// TIA Portal V17 export
// export: Created 2023-02-14T02:49:31.079512Z, ExportSetting WithDefaults, DisplayName Totally Integrated Automation Portal, DisplayVersion V17, DisplayName TIA Portal Openness, DisplayVersion V17, DisplayName TIA Portal Teamcenter Gateway, DisplayVersion V17, DisplayName TIA Portal Version Control Interface, DisplayVersion V17, DisplayName SINAMICS Startdrive Advanced, DisplayVersion V17, DisplayName SINAMICS Startdrive G130, G150, S120, S150, SINAMICS MV, S210, DisplayVersion V17, DisplayName SINAMICS Startdrive G110M, G120, G120C, G120D, G120P, G115D, DisplayVersion V17, DisplayName STEP 7 Professional, DisplayVersion V17, DisplayName STEP 7 Safety, DisplayVersion V17, DisplayName WinCC Professional, DisplayVersion V17
DATA_BLOCK "IO_Valve_Storage_DB"   // DB11
VERSION : 0.1
// stored: AutoNumber true, DBAccessibleFromOPCUA true, DBAccessibleFromWebserver true, InstanceOfName IO_Valve_Storage, InstanceOfType FB
"IO_Valve_Storage"
   // VAR_INPUT
   //    lock : Bool;
   //    Init : Bool;
   //    Reset : Bool;
   // END_VAR
   // VAR
   //    "AV-23.01" { S7_SetPoint := 'True'} : "Valve";
   //    "AV-23.02" { S7_SetPoint := 'True'} : "Valve";
   //    "AV-23.03" { S7_SetPoint := 'True'} : "Valve";
   //    "AV-23.04" { S7_SetPoint := 'True'} : "Valve";
   //    "AV-23.05" { S7_SetPoint := 'True'} : "Valve";
   //    "AV-23.06" { S7_SetPoint := 'True'} : "Valve";
   //    "AV-23.07" { S7_SetPoint := 'True'} : "Valve";
   //    "AV-23.08" { S7_SetPoint := 'True'} : "Valve";
   //    "AV-24.01" { S7_SetPoint := 'True'} : "Valve";
   //    "AV-24.02" { S7_SetPoint := 'True'} : "Valve";
   //    "AV-24.03" { S7_SetPoint := 'True'} : "Valve";
   //    "AV-24.04" { S7_SetPoint := 'True'} : "Valve";
   //    "AV-24.05" { S7_SetPoint := 'True'} : "Valve";
   //    "AV-24.06" { S7_SetPoint := 'True'} : "Valve";
   //    "AV-24.13" { S7_SetPoint := 'True'} : "Valve";
   //    "AV-24.14" { S7_SetPoint := 'True'} : "Valve";
   //    "AV-29.01" { S7_SetPoint := 'True'} : "Valve";
   //    "AV-29.02" { S7_SetPoint := 'True'} : "Valve";
   //    "AV-29.03" { S7_SetPoint := 'True'} : "Valve";
   //    "AV-29.04" { S7_SetPoint := 'True'} : "Valve";
   //    "AV-29.06" { S7_SetPoint := 'True'} : "Valve";
   //    "AV-33.01" { S7_SetPoint := 'True'} : "Valve";
   //    "AV-33.02" { S7_SetPoint := 'True'} : "Valve";
   //    "AV-33.03" { S7_SetPoint := 'True'} : "Valve";
   //    "AV-33.04" { S7_SetPoint := 'True'} : "Valve";
   //    "AV-33.05" { S7_SetPoint := 'True'} : "Valve";
   //    "AV-33.06" { S7_SetPoint := 'True'} : "Valve";
   //    "AV-33.07" { S7_SetPoint := 'True'} : "Valve";
   //    "AV-33.08" { S7_SetPoint := 'True'} : "Valve";
   //    "AV-33.09" { S7_SetPoint := 'True'} : "Valve";
   //    "AV-33.10" { S7_SetPoint := 'True'} : "Valve";
   //    "AV-33.11" { S7_SetPoint := 'True'} : "Valve";
   //    "AV-34.01" { S7_SetPoint := 'True'} : "Valve";
   //    "AV-34.02" { S7_SetPoint := 'True'} : "Valve";
   //    "AV-34.03" { S7_SetPoint := 'True'} : "Valve";
   //    "AV-34.04" { S7_SetPoint := 'True'} : "Valve";
   //    "AV-34.05" { S7_SetPoint := 'True'} : "Valve";
   //    "AV-34.06" { S7_SetPoint := 'True'} : "Valve";
   //    "AV-34.07" { S7_SetPoint := 'True'} : "Valve";
   //    "AV-34.08" { S7_SetPoint := 'True'} : "Valve";
   //    "AV-34.09" { S7_SetPoint := 'True'} : "Valve";
   //    "AV-34.10" { S7_SetPoint := 'True'} : "Valve";
   //    "AV-34.11" { S7_SetPoint := 'True'} : "Valve";
   //    "AV-34.12" { S7_SetPoint := 'True'} : "Valve";
   //    "AV-35.01" { S7_SetPoint := 'True'} : "Valve";
   //    "AV-35.02" { S7_SetPoint := 'True'} : "Valve";
   //    "AV-35.03" { S7_SetPoint := 'True'} : "Valve";
   //    "AV-35.04" { S7_SetPoint := 'True'} : "Valve";
   //    "AV-35.05" { S7_SetPoint := 'True'} : "Valve";
   //    "AV-35.06" { S7_SetPoint := 'True'} : "Valve";
   //    "AV-35.07" { S7_SetPoint := 'True'} : "Valve";
   //    "AV-35.08" { S7_SetPoint := 'True'} : "Valve";
   //    "AV-39.01" { S7_SetPoint := 'True'} : "Valve";
   //    "AV-39.02" { S7_SetPoint := 'True'} : "Valve";
   //    "AV-39.03" { S7_SetPoint := 'True'} : "Valve";
   //    "AV-39.04" { S7_SetPoint := 'True'} : "Valve";
   //    "AV-39.06" { S7_SetPoint := 'True'} : "Valve";
   //    "AV-24.15" { S7_SetPoint := 'True'} : "Valve";
   //    "AV-24.16" { S7_SetPoint := 'True'} : "Valve";
   //    "AV-79.01" { S7_SetPoint := 'True'} : "Valve";
   //    "AV-79.02" { S7_SetPoint := 'True'} : "Valve";
   //    "AV-79.03" { S7_SetPoint := 'True'} : "Valve";
   //    "AV-79.04" { S7_SetPoint := 'True'} : "Valve";
   //    "AV-79.05" { S7_SetPoint := 'True'} : "Valve";
   //    "AV-79.06" { S7_SetPoint := 'True'} : "Valve";
   //    "AV-79.07" { S7_SetPoint := 'True'} : "Valve";
   //    "AV-79.08" { S7_SetPoint := 'True'} : "Valve";
   //    "AV-79.09" { S7_SetPoint := 'True'} : "Valve";
   //    "AV-79.10" { S7_SetPoint := 'True'} : "Valve";
   //    "AV-79.13" { S7_SetPoint := 'True'} : "Valve";
   //    "AV-79.14" { S7_SetPoint := 'True'} : "Valve";
   //    "AV-79.15" { S7_SetPoint := 'True'} : "Valve";
   //    "AV-79.16" { S7_SetPoint := 'True'} : "Valve";
   //    "AV-79.17" { S7_SetPoint := 'True'} : "Valve";
   //    "AV-81.01" { S7_SetPoint := 'True'} : "Valve";
   //    "AV-81.02" { S7_SetPoint := 'True'} : "Valve";
   //    "AV-81.03" { S7_SetPoint := 'True'} : "Valve";
   //    "AV-81.04" { S7_SetPoint := 'True'} : "Valve";
   //    "AV-81.05" { S7_SetPoint := 'True'} : "Valve";
   //    "AV-81.06" { S7_SetPoint := 'True'} : "Valve";
   //    "AV-81.07" { S7_SetPoint := 'True'} : "Valve";
   //    "AV-81.08" { S7_SetPoint := 'True'} : "Valve";
   //    "AV-81.09" { S7_SetPoint := 'True'} : "Valve";
   //    "AV-81.10" { S7_SetPoint := 'True'} : "Valve";
   //    "AV-81.12" { S7_SetPoint := 'True'} : "Valve";
   //    "AV-81.13" { S7_SetPoint := 'True'} : "Valve";
   //    "AV-81.14" { S7_SetPoint := 'True'} : "Valve";
   //    "AV-85.01" { S7_SetPoint := 'True'} : "Valve";
   //    "AV-85.02" { S7_SetPoint := 'True'} : "Valve";
   //    "AV-85.03" { S7_SetPoint := 'True'} : "Valve";
   //    "AV-85.04" { S7_SetPoint := 'True'} : "Valve";
   //    "AV-85.13" { S7_SetPoint := 'True'} : "Valve";
   //    "AV-85.12" { S7_SetPoint := 'True'} : "Valve";
   //    "AV-85.14" { S7_SetPoint := 'True'} : "Valve";
   //    "AV-85.15" { S7_SetPoint := 'True'} : "Valve";
   //    "AV-85.05" { S7_SetPoint := 'True'} : "Valve";
   //    "AV-85.06" { S7_SetPoint := 'True'} : "Valve";
   //    "AV-85.16" { S7_SetPoint := 'True'} : "Valve";
   //    "AV-85.17" { S7_SetPoint := 'True'} : "Valve";
   //    "AV-85.18" { S7_SetPoint := 'True'} : "Valve";
   //    "AV-85.09" { S7_SetPoint := 'True'} : "Valve";
   //    "AV-85.08" { S7_SetPoint := 'True'} : "Valve";
   //    "AV-85.10" { S7_SetPoint := 'True'} : "Valve";
   //    "AV-85.11" { S7_SetPoint := 'True'} : "Valve";
   //    "AV-84.05" { S7_SetPoint := 'True'} : "Valve";
   //    "AV-84.06" { S7_SetPoint := 'True'} : "Valve";
   //    "AV-84.07" { S7_SetPoint := 'True'} : "Valve";
   //    "AV-84.08" { S7_SetPoint := 'True'} : "Valve";
   //    "AV-84.09" { S7_SetPoint := 'True'} : "Valve";
   //    "AV-84.10" { S7_SetPoint := 'True'} : "Valve";
   //    "AV-84.12" { S7_SetPoint := 'True'} : "Valve";
   //    "AV-84.13" { S7_SetPoint := 'True'} : "Valve";
   //    "AV-84.14" { S7_SetPoint := 'True'} : "Valve";
   //    "AV-24.09" { S7_SetPoint := 'True'} : "Valve";
   //    "AV-24.17" { S7_SetPoint := 'True'} : "Valve";
   //    "AV-24.18" { S7_SetPoint := 'True'} : "Valve";
   //    "AV-24.19" { S7_SetPoint := 'True'} : "Valve";
   //    "AV-24.20" { S7_SetPoint := 'True'} : "Valve";
   //    "AV-24.21" { S7_SetPoint := 'True'} : "Valve";
   //    "AV-24.22" { S7_SetPoint := 'True'} : "Valve";
   //    "AV-24.23" { S7_SetPoint := 'True'} : "Valve";
   //    "AV-24.24" { S7_SetPoint := 'True'} : "Valve";
   //    "AV-79.21" { S7_SetPoint := 'True'} : "Valve";
   //    "AV-79.18" { S7_SetPoint := 'True'} : "Valve";
   //    "AV-79.19" { S7_SetPoint := 'True'} : "Valve";
   //    "AV-79.20" { S7_SetPoint := 'True'} : "Valve";
   // END_VAR
BEGIN
END_DATA_BLOCK
